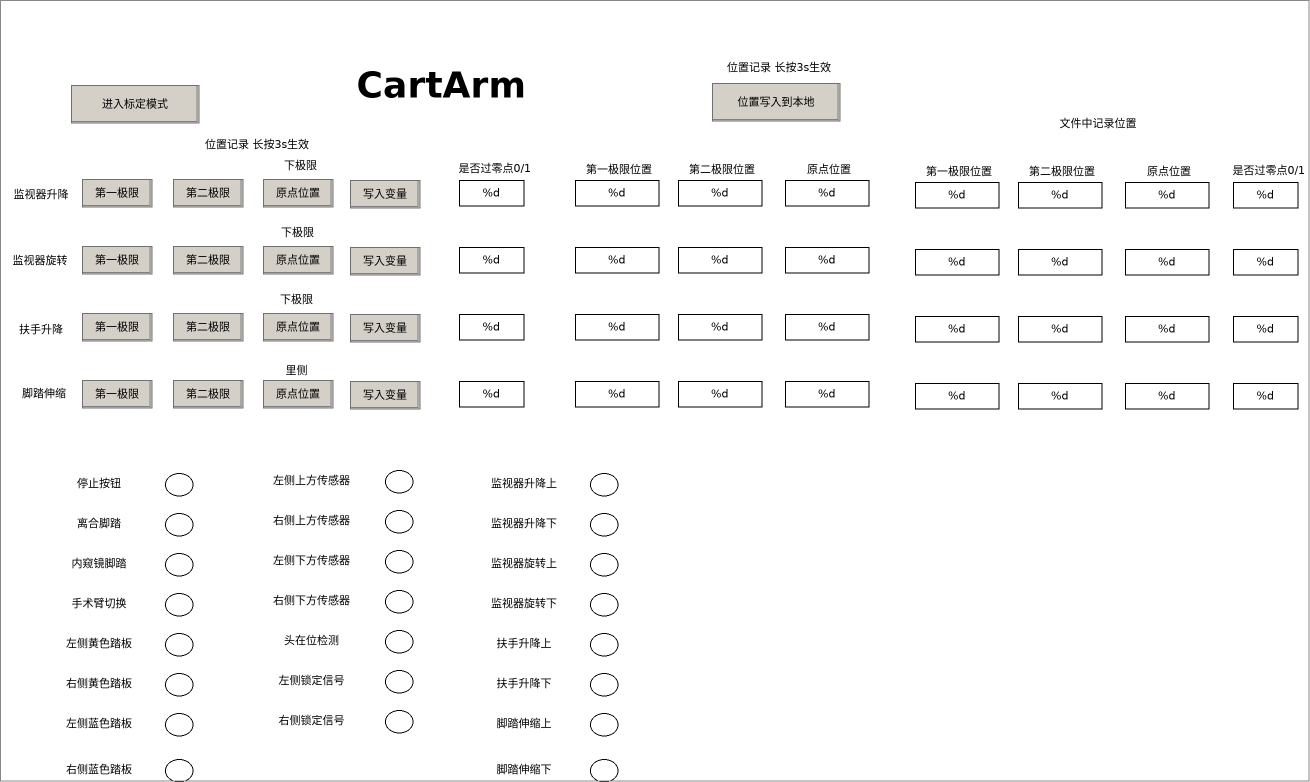
VISUALIZATION carCail  // 1310x782
    Button (71,85 128x38), "进入标定模式", colour toggle: GVL_armCali.g_cartEnterCaliMode
        toggle GVL_armCali.g_cartEnterCaliMode
    Button (82,179 70x28), "第一极限", colour toggle: GVL_armCali.g_linkEncFristCaliTriggerOfCart[1]
        tap GVL_armCali.g_linkEncFristPosCaliOfCart[1]
    Button (173,179 70x28), "第二极限", colour toggle: GVL_armCali.g_linkEncSecondCaliTriggerOfCart[1]
        tap GVL_armCali.g_linkEncSecondPosCaliOfCart[1]
    Rectangle (459,180 65x26), "%d", text variable: GVL_armCali.g_linkZeroCrossOrNotOfCart[1]
    Label (454,157 82x23), "是否过零点0/1"
    Rectangle (575,180 84x26), "%d", text variable: GVL_armCali.g_linkLimitFristPosOfCart[1]
    Label (578,158 82x23), "第一极限位置"
    Rectangle (678,180 84x26), "%d", text variable: GVL_armCali.g_linkLimitSecondPosOfCart[1]
    Label (681,158 82x23), "第二极限位置"
    Label (182,133 150x23), "位置记录 长按3s生效"
    Rectangle (785,180 84x26), "%d", text variable: GVL_armCali.g_linkHomePosOfCart[1]
    Label (788,158 82x23), "原点位置"
    Button (263,179 70x28), "原点位置", colour toggle: GVL_armCali.g_linkEncHomePosCaliTriggerOfCart[1]
        tap GVL_armCali.g_linkEncHomePosCaliOfCart[1]
    Button (82,246 70x28), "第一极限", colour toggle: GVL_armCali.g_linkEncFristCaliTriggerOfCart[2]
        tap GVL_armCali.g_linkEncFristPosCaliOfCart[2]
    Button (173,246 70x28), "第二极限", colour toggle: GVL_armCali.g_linkEncSecondCaliTriggerOfCart[2]
        tap GVL_armCali.g_linkEncSecondPosCaliOfCart[2]
    Rectangle (459,247 65x26), "%d", text variable: GVL_armCali.g_linkZeroCrossOrNotOfCart[2]
    Rectangle (575,247 84x26), "%d", text variable: GVL_armCali.g_linkLimitFristPosOfCart[2]
    Rectangle (678,247 84x26), "%d", text variable: GVL_armCali.g_linkLimitSecondPosOfCart[2]
    Rectangle (785,247 84x26), "%d", text variable: GVL_armCali.g_linkHomePosOfCart[2]
    Button (263,246 70x28), "原点位置", colour toggle: GVL_armCali.g_linkEncHomePosCaliTriggerOfCart[2]
        tap GVL_armCali.g_linkEncHomePosCaliOfCart[2]
    Button (82,313 70x28), "第一极限", colour toggle: GVL_armCali.g_linkEncFristCaliTriggerOfCart[3]
        tap GVL_armCali.g_linkEncFristPosCaliOfCart[3]
    Button (173,313 70x28), "第二极限", colour toggle: GVL_armCali.g_linkEncSecondCaliTriggerOfCart[3]
        tap GVL_armCali.g_linkEncSecondPosCaliOfCart[3]
    Rectangle (459,314 65x26), "%d", text variable: GVL_armCali.g_linkZeroCrossOrNotOfCart[3]
    Rectangle (575,314 84x26), "%d", text variable: GVL_armCali.g_linkLimitFristPosOfCart[3]
    Rectangle (678,314 84x26), "%d", text variable: GVL_armCali.g_linkLimitSecondPosOfCart[3]
    Rectangle (785,314 84x26), "%d", text variable: GVL_armCali.g_linkHomePosOfCart[3]
    Button (263,313 70x28), "原点位置", colour toggle: GVL_armCali.g_linkEncHomePosCaliTriggerOfCart[3]
        tap GVL_armCali.g_linkEncHomePosCaliOfCart[3]
    Button (82,380 70x28), "第一极限", colour toggle: GVL_armCali.g_linkEncFristCaliTriggerOfCart[4]
        tap GVL_armCali.g_linkEncFristPosCaliOfCart[4]
    Button (173,380 70x28), "第二极限", colour toggle: GVL_armCali.g_linkEncSecondCaliTriggerOfCart[4]
        tap GVL_armCali.g_linkEncSecondPosCaliOfCart[4]
    Rectangle (459,381 65x26), "%d", text variable: GVL_armCali.g_linkZeroCrossOrNotOfCart[4]
    Rectangle (575,381 84x26), "%d", text variable: GVL_armCali.g_linkLimitFristPosOfCart[4]
    Rectangle (678,381 84x26), "%d", text variable: GVL_armCali.g_linkLimitSecondPosOfCart[4]
    Rectangle (785,381 84x26), "%d", text variable: GVL_armCali.g_linkHomePosOfCart[4]
    Button (263,380 70x28), "原点位置", colour toggle: GVL_armCali.g_linkEncHomePosCaliTriggerOfCart[4]
        tap GVL_armCali.g_linkEncHomePosCaliOfCart[4]
    Rectangle (915,182 84x26), "%d", text variable: GVL_CartJointCaliData.g_minLinkEncoder[1]
    Label (918,160 82x23), "第一极限位置"
    Rectangle (1018,182 84x26), "%d", text variable: GVL_CartJointCaliData.g_maxLinkEncoder[1]
    Label (1021,160 82x23), "第二极限位置"
    Rectangle (1125,182 84x26), "%d", text variable: GVL_CartJointCaliData.g_caliLinkEncoder[1]
    Label (1128,160 82x23), "原点位置"
    Rectangle (915,249 84x26), "%d", text variable: GVL_CartJointCaliData.g_minLinkEncoder[2]
    Rectangle (1018,249 84x26), "%d", text variable: GVL_CartJointCaliData.g_maxLinkEncoder[2]
    Rectangle (1125,249 84x26), "%d", text variable: GVL_CartJointCaliData.g_caliLinkEncoder[2]
    Rectangle (915,316 84x26), "%d", text variable: GVL_CartJointCaliData.g_minLinkEncoder[3]
    Rectangle (1018,316 84x26), "%d", text variable: GVL_CartJointCaliData.g_maxLinkEncoder[3]
    Rectangle (1125,316 84x26), "%d", text variable: GVL_CartJointCaliData.g_caliLinkEncoder[3]
    Rectangle (915,383 84x26), "%d", text variable: GVL_CartJointCaliData.g_minLinkEncoder[4]
    Rectangle (1018,383 84x26), "%d", text variable: GVL_CartJointCaliData.g_maxLinkEncoder[4]
    Rectangle (1125,383 84x26), "%d", text variable: GVL_CartJointCaliData.g_caliLinkEncoder[4]
    Rectangle (1233,182 65x26), "%d", text variable: GVL_CartJointCaliData.g_linkEncZeroCross[1]
    Label (1228,159 82x23), "是否过零点0/1"
    Rectangle (1233,249 65x26), "%d", text variable: GVL_CartJointCaliData.g_linkEncZeroCross[2]
    Rectangle (1233,316 65x26), "%d", text variable: GVL_CartJointCaliData.g_linkEncZeroCross[3]
    Rectangle (1233,383 65x26), "%d", text variable: GVL_CartJointCaliData.g_linkEncZeroCross[4]
    Button (350,180 70x28), "写入变量", colour toggle: GVL_armCali.g_linkPosWriteCaliDataTriggerOfCart[1]
        tap GVL_armCali.g_linkPosWriteCaliDataOfCart[1]
    Button (350,247 70x28), "写入变量", colour toggle: GVL_armCali.g_linkPosWriteCaliDataTriggerOfCart[2]
        tap GVL_armCali.g_linkPosWriteCaliDataOfCart[2]
    Button (350,314 70x28), "写入变量", colour toggle: GVL_armCali.g_linkPosWriteCaliDataTriggerOfCart[3]
        tap GVL_armCali.g_linkPosWriteCaliDataOfCart[3]
    Button (350,381 70x28), "写入变量", colour toggle: GVL_armCali.g_linkPosWriteCaliDataTriggerOfCart[4]
        tap GVL_armCali.g_linkPosWriteCaliDataOfCart[4]
    Label (343,59 197x52), "CartArm"
    Button (712,83 128x38), "位置写入到本地", colour toggle: GVL_armCali.g_caliDataWriteTriggerOfCart
        tap GVL_armCali.g_caliDataWriteOfCart
    Label (704,56 150x23), "位置记录 长按3s生效"
    Label (1023,112 150x23), "文件中记录位置"
    Label (59,472 80x23), "停止按钮"
    Ellipse (165,473 28x23), colour toggle: GVL_IO.g_stopButton
    Label (59,512 80x23), "离合脚踏"
    Ellipse (165,513 28x23), colour toggle: GVL_IO.g_clutchPedal
    Label (59,552 80x23), "内窥镜脚踏"
    Ellipse (165,553 28x23), colour toggle: GVL_IO.g_endoScopePedal
    Label (59,592 80x23), "手术臂切换"
    Ellipse (165,593 28x23), colour toggle: GVL_IO.g_armSwitch
    Label (59,632 80x23), "左侧黄色踏板"
    Ellipse (165,633 28x23), colour toggle: GVL_IO.g_electricCutLeft
    Label (59,672 80x23), "右侧黄色踏板"
    Ellipse (165,673 28x23), colour toggle: GVL_IO.g_electricCutRight
    Label (59,712 80x23), "左侧蓝色踏板"
    Ellipse (165,713 28x23), colour toggle: GVL_IO.g_electricCoagulLeft
    Label (59,758 80x23), "右侧蓝色踏板"
    Ellipse (165,759 28x23), colour toggle: GVL_IO.g_electricCoagulRight
    Label (264,469 95x23), "左侧上方传感器"
    Ellipse (385,470 28x23), colour toggle: GVL_IO.g_electricCutLeftSensor
    Label (264,509 95x23), "右侧上方传感器"
    Ellipse (385,510 28x23), colour toggle: GVL_IO.g_electricCutRightSensor
    Label (264,549 95x23), "左侧下方传感器"
    Ellipse (385,550 28x23), colour toggle: GVL_IO.g_electricCoagulLeftSensor
    Label (264,589 95x23), "右侧下方传感器"
    Ellipse (385,590 28x23), colour toggle: GVL_IO.g_electricCoagulRightSensor
    Label (264,629 95x23), "头在位检测"
    Ellipse (385,630 28x23), colour toggle: GVL_IO.g_surgonHeadIn
    Label (264,669 95x23), "左侧锁定信号"
    Ellipse (385,670 28x23), colour toggle: GVL_IO.g_cartLockSignalLeft
    Label (264,709 95x23), "右侧锁定信号"
    Ellipse (385,710 28x23), colour toggle: GVL_IO.g_cartLockSignalRight
    Label (484,472 80x23), "监视器升降上"
    Ellipse (590,473 28x23), colour toggle: GVL_IO.g_cartJointCtrl[1]
    Label (484,512 80x23), "监视器升降下"
    Ellipse (590,513 28x23), colour toggle: GVL_IO.g_cartJointCtrl[2]
    Label (484,552 80x23), "监视器旋转上"
    Ellipse (590,553 28x23), colour toggle: GVL_IO.g_cartJointCtrl[4]
    Label (484,592 80x23), "监视器旋转下"
    Ellipse (590,593 28x23), colour toggle: GVL_IO.g_cartJointCtrl[3]
    Label (484,632 80x23), "扶手升降上"
    Ellipse (590,633 28x23), colour toggle: GVL_IO.g_cartJointCtrl[5]
    Label (484,672 80x23), "扶手升降下"
    Ellipse (590,673 28x23), colour toggle: GVL_IO.g_cartJointCtrl[6]
    Label (484,712 80x23), "脚踏伸缩上"
    Ellipse (590,713 28x23), colour toggle: GVL_IO.g_cartJointCtrl[8]
    Label (484,758 80x23), "脚踏伸缩下"
    Ellipse (590,759 28x23), colour toggle: GVL_IO.g_cartJointCtrl[7]
    Label (270,155 61x21), "下极限"
    Label (266,289 61x21), "下极限"
    Label (266,360 61x21), "里侧"
    Label (5,184 72x21), "监视器升降"
    Label (4,250 72x21), "监视器旋转"
    Label (5,319 72x21), "扶手升降"
    Label (8,383 72x21), "脚踏伸缩"
    Label (267,222 61x21), "下极限"
END_VISUALIZATION

(* stored: Version 1.1.0.1, ProductVersion 3.1.4024.11
   Visu carCail: Id {761fe35a-e76f-46c0-8e2a-58082bc85c4b} *)
